Staubli VAL3: Wizard.dtx

bool bActiveLevel = true
bool bForDisplay = true
bool bIsScara = true
bool bStopRead
bool bUseLatch = true
dio doClock = {link=BasicIO-1\%Q0}
public mdesc mNomSpeed = {rmax=9999, blend=off}
mdesc mSlow = {tmax=100, blend=off, leave=5, reach=5}
num nLanguage = 1
num nLblPosX
num nLblPosY
num nMANUAL = 1
num nMANUAL_HOLD = 6
num nMAXLANG = 1
num nMotionError
num nPagePosX
num nPagePosY
num nScaleFact[2]
num nStackSize = 5
num nTxtMaxVal
num nTxtMinVal
num nTxtPosX
num nTxtPosY
num nVIDEOCUSTOM = 2
num nVIDEOINVERSED = 1
num nVIDEONORMAL
string sCaption[12]
  [0] = "EncoderLib: "
  [1] = "Detect Lib: "
  [2] = "BufferSize: "
  [3] = "ScaleFact : "
  [4] = "Height    :"
  [5] = "ThruUpLim :"
  [6] = "ThruDwnLim:"
  [7] = "MatchTol: "
  [8] = "ClkSignal:"
  [9] = "ClkPeriod: "
  [10] = "LockDist : "
  [11] = "Enable Log:"
string sConveyorFile = "cvIn"
string sDOutputsList[18]
  [0] = "none"
  [1] = "bOut0"
  [2] = "bOut1"
  [3] = "bOut10"
  [4] = "bOut11"
  [5] = "bOut12"
  [6] = "bOut13"
  [7] = "bOut14"
  [8] = "bOut15"
  [9] = "bOut2"
  [10] = "bOut3"
  [11] = "bOut4"
  [12] = "bOut5"
  [13] = "bOut6"
  [14] = "bOut7"
  [15] = "bOut8"
  [16] = "bOut9"
  [17] = "fOut0"
string sErrorMessage = "The detection library Disk://Tracking\Detections\Cognex1 could not be loaded because of error code 12 "
string sGenericDet = "GenericDetect"
string sGenericEnc = "GenericEnc"
string sGeometryLib = "GeometryRS"
string sItemList[7]
  [0] = "Cognex1"
  [1] = "Cognex2"
  [2] = "PointGrey"
  [3] = "Sensor1"
  [4] = "Sensor2"
  [5] = "Socket1"
  [6] = "Socket2"
string sLangFile[2]
  [1] = "chinese"
string sUnwantDOutputs[5]
  [0] = "world flange"
  [1] = "b2Out0 b2Out1 b2Out2 b2Out3 b2Out4 b2Out5 b2Out6 b2Out7 b2Out8 b2Out9 b2Out10 b2Out11 b2Out12 b2Out13 b2Out14 b2Out15"
  [2] = "cDout0 cDout1 cDout2 cDout3 cDout4 cDout5 cDout6 cDout7"
  [3] = "mOut0 mOut1 mOut2 mOut3 mOut4 mOut5 mOut6 mOut7 mOut8 mOut9 mOut10 mOut11 mOut12 mOut13 mOut14 mOut15"
  [4] = "mOut16 mOut17 mOut18 mOut19 mOut20 mOut21 mOut22 mOut23 mOut24 mOut25 mOut26 mOut27 mOut28 mOut29 mOut30 mOut31"
tool tPointer = {z=130, fatherId=flange[0], ioLink=valve1}
